// TIA Portal V18 export
DATA_BLOCK "DATA"   // DB2
{ S7_Optimized_Access := 'TRUE' }
VERSION : 0.1
// stored: AutoNumber true, DBAccessibleFromOPCUA true, DBAccessibleFromWebserver true, IsOnlyStoredInLoadMemory false, IsRetainMemResEnabled false, IsWriteProtectedInAS false, MemoryReserve 100
   VAR
      Str : String := '0+252+65526+5000+955+54+100+566';
      Str_1 : String[4];
      Val_1 : DInt;
      Val_2 : DInt;
      Val_3 : DInt;
   END_VAR
BEGIN
END_DATA_BLOCK
